GLOBALCONSTANTS ISO_NETEVENT_e (* Global constants for network management event types *)
  (* Standard: 61499-1 *)
  (* Version 1.0, 2025-10-18, franz *)
  PACKAGE isobus::pgn;
  VAR_GLOBAL CONSTANT
    Isonet_MemberActive : USINT := 0;
    Isonet_MemberAddressConflict : USINT := 1;
    Isonet_MemberInactive : USINT := 2;
    Isonet_MemberNewAddress : USINT := 3;
    Isonet_MemberAddressViolation : USINT := 4;
    Isonet_MemberAdd : USINT := 5;
    Isonet_MemberRemove : USINT := 6;
    Isonet_HsiActive : USINT := 7;
    Isonet_HsiInactive : USINT := 8;
    Isonet_Last : USINT := 9;
  END_VAR
END_GLOBALCONSTANTS
